(* PLC project Unnamed, Unknown Unnamed 1 *)
(* stored: creationDateTime 2022-10-03T20:09:30, modificationDateTime 2022-10-07T01:01:19 *)

PROGRAM trafficSignl
  VAR
    RED1 AT %QX100.0 : BOOL;
    YELLOW1 AT %QX100.1 : BOOL;
    GREEN1 AT %QX100.2 : BOOL;
    RED2 AT %QX0.0 : BOOL := true;
    YELLOW2 AT %QX0.1 : BOOL;
    GREEN2 AT %QX0.2 : BOOL;
    Time_GREEN1 AT %MW0 : INT;
    Time_YELLOW1 AT %MW1 : INT;
    Time_RED1 AT %MW2 : INT;
    Time_GREEN2 AT %MW3 : INT;
    Time_YELLOW2 AT %MW4 : INT;
    Time_RED2 AT %MW5 : INT;
  END_VAR
  VAR
    TON0 : TON;
    TON1 : TON;
    TON2 : TON;
    TON3 : TON;
  END_VAR
  VAR  (* added by the conversion: wires and edge detectors of the diagram *)
    _SUB39_OUT : INT;
    _SUB75_OUT : INT;
  END_VAR

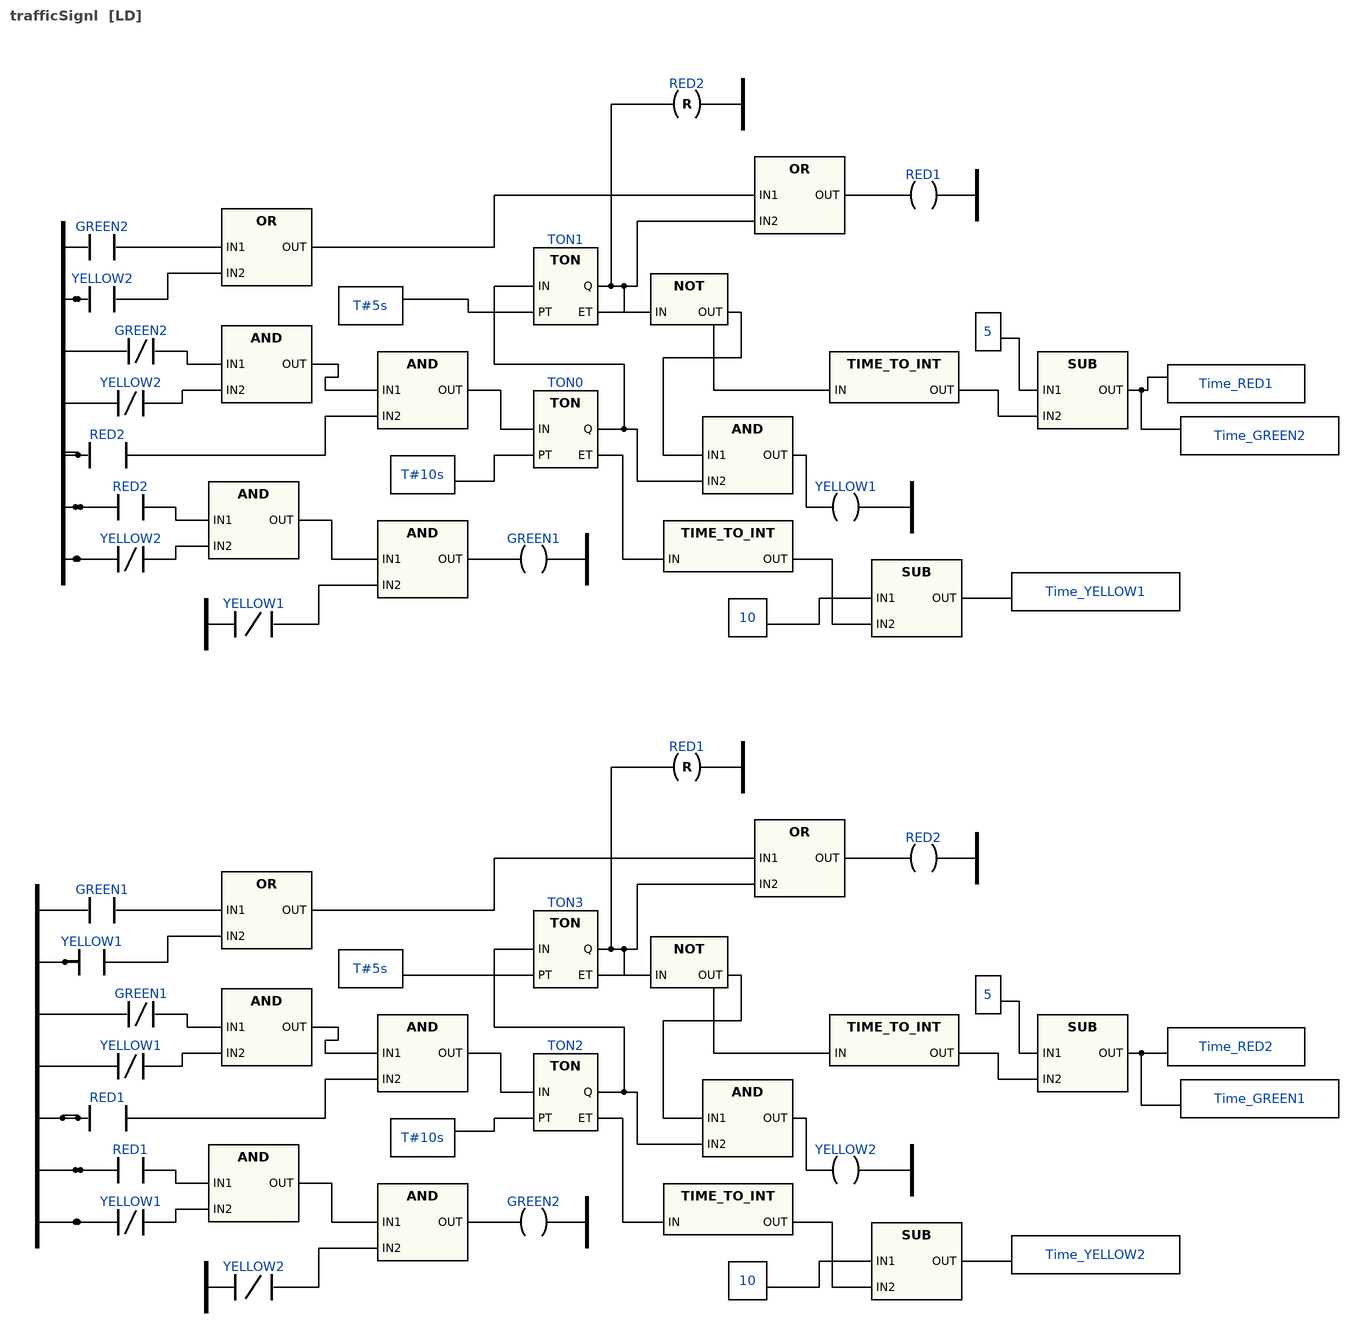
(* LD diagram, written out as Structured Text *)
TON0(IN := NOT GREEN2 AND NOT YELLOW2 AND RED2, PT := T#10s);
TON1(IN := TON0.Q, PT := T#5s);
IF TON1.Q THEN RED2 := FALSE; END_IF;
RED1 := GREEN2 OR YELLOW2 OR TON1.Q;
_SUB39_OUT := 5 - TIME_TO_INT(TON1.ET);
Time_RED1 := _SUB39_OUT;
Time_GREEN2 := _SUB39_OUT;
YELLOW1 := NOT TON1.Q AND TON0.Q;
GREEN1 := RED2 AND NOT YELLOW2 AND NOT YELLOW1;
Time_YELLOW1 := 10 - TIME_TO_INT(TON0.ET);
TON2(IN := NOT GREEN1 AND NOT YELLOW1 AND RED1, PT := T#10s);
TON3(IN := TON2.Q, PT := T#5s);
IF TON3.Q THEN RED1 := FALSE; END_IF;
RED2 := GREEN1 OR YELLOW1 OR TON3.Q;
_SUB75_OUT := 5 - TIME_TO_INT(TON3.ET);
Time_RED2 := _SUB75_OUT;
Time_GREEN1 := _SUB75_OUT;
YELLOW2 := NOT TON3.Q AND TON2.Q;
GREEN2 := RED1 AND NOT YELLOW1 AND NOT YELLOW2;
Time_YELLOW2 := 10 - TIME_TO_INT(TON2.ET);
END_PROGRAM

CONFIGURATION Config0
  RESOURCE Res0 ON PLC
    TASK task0(INTERVAL := T#20ms, PRIORITY := 0);
    PROGRAM instance0 WITH task0 : trafficSignl;
  END_RESOURCE
END_CONFIGURATION
